Staubli VAL3: ChangeCirPoint.pgx

public program ChangeCirPoint(trsf x_trCenter, num x_nDia, trsf& x_trSource, trsf x_trSupport, bool& x_bRes)
  local frame l_fFrame
  local point l_pPoint[3]
begin
  //根据边长和圆心点来修改相应的点。

  x_bRes=false

  if x_nDia<=0
    return
  endIf

  l_pPoint[0].trsf=x_trCenter
  l_pPoint[1].trsf=x_trSource
  l_pPoint[2].trsf=x_trSupport

  link(l_pPoint[0],world)
  link(l_pPoint[1],world)
  link(l_pPoint[2],world)
  link(l_fFrame,world)

  if setFrame(l_pPoint[0],l_pPoint[1],l_pPoint[2],l_fFrame)!=0
    return
  endIf

  l_pPoint[1].trsf=position(l_pPoint[1],l_fFrame)
  l_pPoint[1].trsf.x=x_nDia/2
  link(l_pPoint[1],l_fFrame)
  x_trSource=position(l_pPoint[1],world)
  x_bRes=true

end
